// TIA Portal project "CajaDeLeche" (V14)

(* hardware
DEVICE "S71500/ET200MP-Station_1"  S7-1500 station
   slot 0: "Profilschiene_0"  6ES7 590-1***0-0AA0
   slot 1: "PLC_1"  CPU 1511-1 PN  6ES7 511-1AK00-0AB0  V1.8
   slot 2: "AI 8xU/I/RTD/TC ST_1"  AI 8xU/I/RTD/TC ST  6ES7 531-7KF00-0AB0  V2.0
   slot 3: "AI 8xU/I/RTD/TC ST_2"  AI 8xU/I/RTD/TC ST  6ES7 531-7KF00-0AB0  V2.0
   slot 4: "AI 8xU/I/RTD/TC ST_3"  AI 8xU/I/RTD/TC ST  6ES7 531-7KF00-0AB0  V2.0
   slot 5: "AI 4xU/I/RTD/TC ST_1"  AI 4xU/I/RTD/TC ST  6ES7 531-7QD00-0AB0  V1.0
   slot 6: "DI 32x24VDC BA_1"  DI 32x24VDC BA  6ES7 521-1BL10-0AA0  V1.0
   slot 7: "DI 32x24VDC BA_2"  DI 32x24VDC BA  6ES7 521-1BL10-0AA0  V1.0
   slot 8: "AQ 4xU/I ST_1"  AQ 4xU/I ST  6ES7 532-5HD00-0AB0  V2.1
   slot 9: "DI 16x24VDC BA_1"  DI 16x24VDC BA  6ES7 521-1BH10-0AA0  V1.0
   slot 10: "DQ 32x24VDC/0.5A ST_1"  DQ 32x24VDC/0.5A ST  6ES7 522-1BL00-0AB0  V2.0
   slot 11: "AQ 4xU/I ST_2"  AQ 4xU/I ST  6ES7 532-5HD00-0AB0  V2.1
   slot 12: "AQ 4xU/I ST_3"  AQ 4xU/I ST  6ES7 532-5HD00-0AB0  V2.1
DEVICE "PC-System_2"  SIMATIC PC station
   slot 0: "Estación PC SIMATIC"  Rail  SIMATIC PC-Station  V1.0
      slot 125: "Stationmanager"  Station_Manager  V6.0.4
   slot 1: "HMI_RT_1"  WinCC RT Professional  6AV2 105-0xxxx-xxxx  14.0.1.0
   slot 2: "IE general_1"  IE General  IE_CP  V8.2.0
*)

// ===== PLC "PLC_1"  CPU 1511-1 PN =====

VAR_GLOBAL   // PLC tag table "Standard-Variablentabelle"
   "Tag_1" AT %E0.0 : Bool;
   "Tag_2" AT %A0.0 : Bool;
   "Tag_3" AT %E0.1 : Bool;
   "LCV001" AT %QW0 : Int;
   "FCV001" AT %QW2 : Int;
   "LT001" AT %IW0 : Int;
   "FT001" AT %IW2 : Int;
   "S_Arranque" AT %I56.0 : Bool;
   "S_Parada" AT %I56.1 : Bool;
   "B_Reset" AT %I56.2 : Bool;
   "SD010" AT %I56.3 : Bool;
   "SD020" AT %I56.4 : Bool;   // Detecta la presencia de la caja vacia
   "SD021" AT %I56.5 : Bool;   // Detecta la presencia de la caja cuando se esta llenando
   "Emisor_Cajas" AT %Q8.0 : Bool;
   "MZ020" AT %Q8.1 : Bool;   // Movimiento Eje Z
   "SZ020" AT %Q8.2 : Bool;   // Succion
   "MZ030" AT %Q8.3 : Bool;   // Movimiento Eje Z
   "SZ030" AT %Q8.4 : Bool;   // Succion
   "CINTA1" AT %Q8.5 : Bool;
   "CINTA2" AT %Q8.6 : Bool;
   "CINTA3" AT %Q8.7 : Bool;
   "CINTA4" AT %Q9.0 : Bool;
   "BSTOP1" AT %Q9.1 : Bool;
   "SD030" AT %I56.7 : Bool;   // Detecta la presencia de la caja llena
   "SD031" AT %I57.0 : Bool;   // Detecta la presencia de la caja cuando se esta colocando la tapa
   "SD022" AT %I56.6 : Bool;
   "SD032" AT %I57.1 : Bool;
   "SD040" AT %I57.2 : Bool;
   "BARRERA_IR" AT %IW4 : Int;
   "Tag_4" AT %QB0 : Byte;
   "Tag_5" AT %QB8 : Byte;
   "Tag_6" AT %QB9 : Byte;
   "Tag_7" AT %QB10 : Byte;
   "Display" AT %QW6 : Int;
   "V001" AT %Q11.2 : Bool;
   "WL04" AT %Q11.3 : Bool;
   "BSTOP2" AT %Q9.2 : Bool;
   "LedBajoNivel" AT %Q9.3 : Bool;
   "LedNivelOk" AT %Q9.4 : Bool;
   "LedContador" AT %Q9.5 : Bool;
   "LedFin" AT %Q9.6 : Bool;
   "LedLLenado" AT %Q9.7 : Bool;
   "VPISTON" AT %QW12 : Int;
   "DISPLAY_NIVEL_TANQUE" AT %QW14 : Int;
   "DISPLAY_SET_NIVEL" AT %QW16 : Int;
   "DISPLAY_NUMERO_BOTELLAS" AT %QW18 : Int;
   "DISPLAY_CONTADOR" AT %QW20 : Int;
   "DISPLAY_PID" AT %QW22 : Int;
   "DISPLAY_SETPINT_LITROS" AT %QW24 : Int;
   "P_PISTON" AT %IW8 : Int;
   "POTE_NIVEL" AT %IW10 : Int;
   "POTE_CANTIDAD_BOTELLA" AT %IW12 : Int;
   "POTE_ESTABLECER_LITROS" AT %IW14 : Int;
   "B_Remoto" AT %I57.3 : Bool;
   "B_Local" AT %I57.4 : Bool;
   "B_Formula1" AT %I57.5 : Bool;
   "B_Formula 2" AT %I57.6 : Bool;
END_VAR

VAR_GLOBAL   // PLC tag table "Paletizado"
   "CINTA_SUPERIOR" AT %Q10.0 : Bool;
   "LIMITE_EMPUJADOR" AT %I57.7 : Bool;
   "PALETA" AT %Q10.1 : Bool;
   "EMPUJADOR" AT %Q10.2 : Bool;
   "LIMITE_PLACA" AT %I58.0 : Bool;
   "PLACA" AT %Q10.3 : Bool;
   "EMISOR_PALLET" AT %Q10.4 : Bool;
   "SENSOR_REFLECTIVO_TRASERO" AT %I58.1 : Bool;
   "SENSOR_REFLECTIVO_DELANTERO" AT %I58.2 : Bool;
   "TRANSPORTADOR_DE_RODILLOS_1" AT %Q10.5 : Bool;
   "SENSOR_LIMITE_FRONTAL" AT %I58.3 : Bool;
   "SENSOR_LIMITE_TRASERO" AT %I58.4 : Bool;
   "CADENA_PALETIZADORA" AT %Q10.6 : Bool;
   "ELEVADOR_SUBIR" AT %Q10.7 : Bool;
   "ELEVADOR_BAJAR" AT %Q11.0 : Bool;
   "ELEVADOR_MOVER_AL_LIMITE" AT %Q11.1 : Bool;
   "SENSOR_CONTADOR" AT %I58.5 : Bool;
   "JUNTAR" AT %Q11.4 : Bool;
   "SENSOR_LIMITE_ELEVADOR" AT %I58.6 : Bool;
END_VAR

DATA_BLOCK "Datos"   // DB1
{ S7_Optimized_Access := 'TRUE' }
VERSION : 0.1
   VAR
      Lecturas : Struct
         "LT001 (mm)" : Real;
         "VT001(L)" : Int;
         "LT001F (mm)" : Real;
         NCAJAS : Int;
         "FT001 (m3/s)" : Real;
         "Posicion (cm)" : Real;
         "Velocidad (cm/s)" : Int;
      END_STRUCT;
      "Set Point" : Struct
         SetPoint_Litros : Int := 1000;
         SetPoint_Cantidad : Int := 20;
         SetPoint_LCV001 : Int := 2000;
      END_STRUCT;
      Dispositivos : Struct
         Tanque : Struct
            L_Maximo : Real := 3000.0;
            L_Minimo : Real;
         END_STRUCT;
      END_STRUCT;
      Constantes : Struct
         A_Lectura_Max_10V : Int := 27648;
         A_Lectura_Min_0V : Int;
      END_STRUCT;
      Etiquetas : Struct
         Emisor : Struct
            Marca : Array[0..10] of Bool;
         END_STRUCT;
         LlenarBotella : Bool;
         Reset : Bool;
         Proceso : Struct
            On : Bool;
            Off : Bool;
         END_STRUCT;
      END_STRUCT;
   END_VAR
BEGIN
END_DATA_BLOCK

DATA_BLOCK "Tableros_DB"   // DB4
{ S7_Optimized_Access := 'TRUE' }
VERSION : 0.1
// stored: InstanceOfName Tableros
"Tableros"
BEGIN
END_DATA_BLOCK

DATA_BLOCK "Paletizado_DB"   // DB5
{ S7_Optimized_Access := 'TRUE' }
VERSION : 0.1
// stored: InstanceOfName Paletizado
"Paletizado"
BEGIN
END_DATA_BLOCK

DATA_BLOCK "Integrador_DB"   // DB14
{ S7_Optimized_Access := 'TRUE' }
VERSION : 0.1
// stored: InstanceOfName Integrador
"Integrador"
BEGIN
END_DATA_BLOCK

DATA_BLOCK "Proceso_Linea_DB"   // DB22
{ S7_Optimized_Access := 'TRUE' }
VERSION : 0.1
// stored: InstanceOfName Proceso_Linea
"Proceso_Linea"
BEGIN
END_DATA_BLOCK

// folder: System blocks/Program resources

DATA_BLOCK "Empujador_retardo"   // DB6
{ S7_Optimized_Access := 'TRUE' }
AUTHOR : Simatic
FAMILY : IEC
NAME : IEC_TMR
VERSION : 1.0
// stored: InstanceOfName IEC_TIMER
"IEC_TIMER"
BEGIN
END_DATA_BLOCK

DATA_BLOCK "Tiempo_Emisor_Pallet"   // DB7
{ S7_Optimized_Access := 'TRUE' }
AUTHOR : Simatic
FAMILY : IEC
NAME : IEC_TMR
VERSION : 1.0
// stored: InstanceOfName IEC_TIMER
"IEC_TIMER"
BEGIN
END_DATA_BLOCK

DATA_BLOCK "RETARDO"   // DB8
{ S7_Optimized_Access := 'TRUE' }
AUTHOR : Simatic
FAMILY : IEC
NAME : IEC_TMR
VERSION : 1.0
// stored: InstanceOfName IEC_TIMER
"IEC_TIMER"
BEGIN
END_DATA_BLOCK

DATA_BLOCK "BAJAR"   // DB9
{ S7_Optimized_Access := 'TRUE' }
AUTHOR : Simatic
FAMILY : IEC
NAME : IEC_TMR
VERSION : 1.0
// stored: InstanceOfName IEC_TIMER
"IEC_TIMER"
BEGIN
END_DATA_BLOCK

DATA_BLOCK "Contador_Cajas_Paletizadora_A"   // DB10
{ S7_Optimized_Access := 'TRUE' }
AUTHOR : Simatic
FAMILY : IEC
NAME : CNTR
VERSION : 1.0
// stored: InstanceOfName IEC_COUNTER
"IEC_COUNTER"
BEGIN
END_DATA_BLOCK

DATA_BLOCK "Contar_3_Filas"   // DB11
{ S7_Optimized_Access := 'TRUE' }
AUTHOR : Simatic
FAMILY : IEC
NAME : CNTR
VERSION : 1.0
// stored: InstanceOfName IEC_COUNTER
"IEC_COUNTER"
BEGIN
END_DATA_BLOCK

DATA_BLOCK "iee"   // DB12
{ S7_Optimized_Access := 'TRUE' }
AUTHOR : Simatic
FAMILY : IEC
NAME : CNTR
VERSION : 1.0
// stored: InstanceOfName IEC_COUNTER
"IEC_COUNTER"
BEGIN
END_DATA_BLOCK

DATA_BLOCK "RETARDO_BAJAR_PALLET"   // DB13
{ S7_Optimized_Access := 'TRUE' }
AUTHOR : Simatic
FAMILY : IEC
NAME : IEC_TMR
VERSION : 1.0
// stored: InstanceOfName IEC_TIMER
"IEC_TIMER"
BEGIN
END_DATA_BLOCK

DATA_BLOCK "Emisor"   // DB18
{ S7_Optimized_Access := 'TRUE' }
AUTHOR : Simatic
FAMILY : IEC
NAME : IEC_TMR
VERSION : 1.0
// stored: InstanceOfName IEC_TIMER
"IEC_TIMER"
BEGIN
END_DATA_BLOCK

DATA_BLOCK "Ton_ColocacionDeTapa"   // DB19
{ S7_Optimized_Access := 'TRUE' }
AUTHOR : Simatic
FAMILY : IEC
NAME : IEC_TMR
VERSION : 1.0
// stored: InstanceOfName IEC_TIMER
"IEC_TIMER"
BEGIN
END_DATA_BLOCK

DATA_BLOCK "Contador_BotellasEmitidas"   // DB21
{ S7_Optimized_Access := 'TRUE' }
AUTHOR : Simatic
FAMILY : IEC
NAME : CNTR
VERSION : 1.0
// stored: InstanceOfName IEC_COUNTER
"IEC_COUNTER"
BEGIN
END_DATA_BLOCK

DATA_BLOCK "IEC_Timer_0_DB_1"   // DB26
{ S7_Optimized_Access := 'TRUE' }
AUTHOR : Simatic
FAMILY : IEC
NAME : IEC_TMR
VERSION : 1.0
// stored: InstanceOfName IEC_TIMER
"IEC_TIMER"
BEGIN
END_DATA_BLOCK

// folder: (top level)

FUNCTION_BLOCK "Tableros"   // FB1, LAD
{ S7_Optimized_Access := 'TRUE' }
VERSION : 0.1
   VAR_INPUT
      Local : Bool;
      Remoto : Bool;
      "Formula 1" : Bool;
      "Formula 2" : Bool;
      Nivel : Real;
      "Nro Botellas" : Real;
      "mL por Botella" : Real;
   END_VAR
   VAR_OUTPUT
      Display_Nivel_Actual : Int;
      Display_Nivel_Seteado : Int;
      Display_Nro_Botellas : Int;
      Display_Contador : Int;
      Display_ml : Int;
      Display_PID : Int;
   END_VAR
   VAR
      "Nivel Temp" : Int;
      "Numero Temp" : Int;
      "mL Temp" : Int;
   END_VAR
BEGIN

REGION Network 1
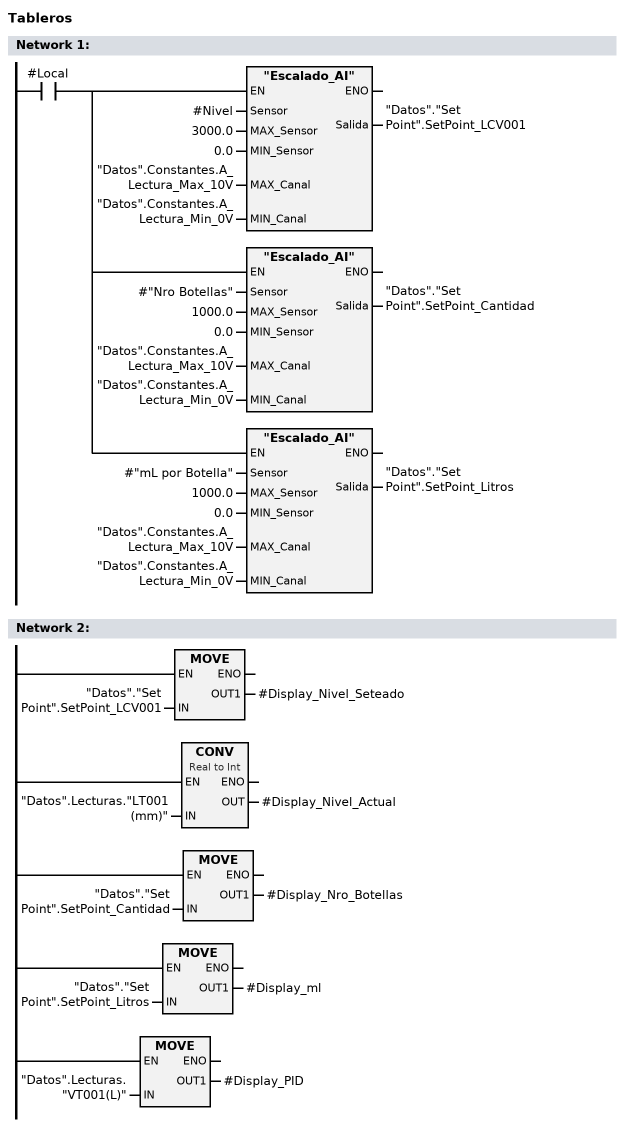
   RUNG wire#powerrail
      Contact( #Local )
      wire#w1
      "Escalado_AI"(Sensor := #Nivel, MAX_Sensor := 3000.0, MIN_Sensor := 0.0, MAX_Canal := "Datos".Constantes.A_Lectura_Max_10V, MIN_Canal := "Datos".Constantes.A_Lectura_Min_0V, Salida => "Datos"."Set Point".SetPoint_LCV001)
   END_RUNG
   RUNG wire#w1
      "Escalado_AI"(Sensor := #"Nro Botellas", MAX_Sensor := 1000.0, MIN_Sensor := 0.0, MAX_Canal := "Datos".Constantes.A_Lectura_Max_10V, MIN_Canal := "Datos".Constantes.A_Lectura_Min_0V, Salida => "Datos"."Set Point".SetPoint_Cantidad)
   END_RUNG
   RUNG wire#w1
      "Escalado_AI"(Sensor := #"mL por Botella", MAX_Sensor := 1000.0, MIN_Sensor := 0.0, MAX_Canal := "Datos".Constantes.A_Lectura_Max_10V, MIN_Canal := "Datos".Constantes.A_Lectura_Min_0V, Salida => "Datos"."Set Point".SetPoint_Litros)
   END_RUNG
   // the same network as SCL:
   IF #Local THEN
       "Escalado_AI"(Sensor := #Nivel,
                     MAX_Sensor := 3000.0,
                     MIN_Sensor := 0.0,
                     MAX_Canal := "Datos".Constantes.A_Lectura_Max_10V,
                     MIN_Canal := "Datos".Constantes.A_Lectura_Min_0V,
                     Salida => "Datos"."Set Point".SetPoint_LCV001);
       "Escalado_AI"(Sensor := #"Nro Botellas",
                     MAX_Sensor := 1000.0,
                     MIN_Sensor := 0.0,
                     MAX_Canal := "Datos".Constantes.A_Lectura_Max_10V,
                     MIN_Canal := "Datos".Constantes.A_Lectura_Min_0V,
                     Salida => "Datos"."Set Point".SetPoint_Cantidad);
       "Escalado_AI"(Sensor := #"mL por Botella",
                     MAX_Sensor := 1000.0,
                     MIN_Sensor := 0.0,
                     MAX_Canal := "Datos".Constantes.A_Lectura_Max_10V,
                     MIN_Canal := "Datos".Constantes.A_Lectura_Min_0V,
                     Salida => "Datos"."Set Point".SetPoint_Litros);
   END_IF;
END_REGION

REGION Network 2
   RUNG wire#powerrail
      Move(in := "Datos"."Set Point".SetPoint_LCV001, out1 => #Display_Nivel_Seteado)
   END_RUNG
   RUNG wire#powerrail
      { S7_Templates := "[SrcType := Real, DestType := Int]" } Convert(in := "Datos".Lecturas."LT001 (mm)", out => #Display_Nivel_Actual)
   END_RUNG
   RUNG wire#powerrail
      Move(in := "Datos"."Set Point".SetPoint_Cantidad, out1 => #Display_Nro_Botellas)
   END_RUNG
   RUNG wire#powerrail
      Move(in := "Datos"."Set Point".SetPoint_Litros, out1 => #Display_ml)
   END_RUNG
   RUNG wire#powerrail
      Move(in := "Datos".Lecturas."VT001(L)", out1 => #Display_PID)
   END_RUNG
   // the same network as SCL:
   #Display_Nivel_Seteado := "Datos"."Set Point".SetPoint_LCV001;
   #Display_Nivel_Actual := REAL_TO_INT("Datos".Lecturas."LT001 (mm)");
   #Display_Nro_Botellas := "Datos"."Set Point".SetPoint_Cantidad;
   #Display_ml := "Datos"."Set Point".SetPoint_Litros;
   #Display_PID := "Datos".Lecturas."VT001(L)";
END_REGION
END_FUNCTION_BLOCK

FUNCTION_BLOCK "Paletizado"   // FB2, LAD
{ S7_Optimized_Access := 'TRUE' }
VERSION : 0.1
   VAR_INPUT
      ARRANQUE : Bool;
      LIMITE_EMPUJADOR : Bool;
      LIMITE_PLACA : Bool;
      SENSOR_REFLECTIVO_TRASERO : Bool;
      SENSOR_REFLECTIVO_DELANTERO : Bool;
      SENSOR_LIMITE_FRONTAL : Bool;
      SENSOR_LIMITE_TRESERO : Bool;
      SENSOR_CONTADOR : Bool;
      SENSOR_LIMITE_ELEVADOR : Bool;
   END_VAR
   VAR_OUTPUT
      CINTA_SUPERIOR : Bool;
      PALETA : Bool;
      EMPUJADOR : Bool;
      PLACA : Bool;
      EMISOR_PALLET : Bool;
      TRANSPORTADOR_DE_RODILLO : Bool;
      CADENA_PALETIZADORA : Bool;
      ELEVADOR_SUBIR : Bool;
      ELEVADOR_BAJAR : Bool;
      ELEVADOR_MOVER_AL_LIMITE : Bool;
      JUNTAR : Bool;
   END_VAR
   VAR
      Flanco : Array[0..40] of Bool;
      Marcas : Array[0..10] of Bool;
      Marca_Emisor : Array[0..10] of Bool;
      REINICIAR_CONT_A : Bool;
      "Contar 2 CAJAS" : Int;
      FILAS : Bool := true;
      CONTEO_B : Int := 2;
      REINICIAR_CONTEO_B : Bool;
      CONTEO_A : Int := 3;
      REINICIAR_CONTEO_C : Bool;
      BYTES : Byte := 16#0;
      CONTAR_ALTURA_FILAS : Bool;
   END_VAR
   VAR_TEMP   // added for the SCL form of the ladder/FBD networks
      _w1 : Bool;
      _w2 : Bool;
      _w3 : Bool;
      _w4 : Bool;
      _w5 : Bool;
   END_VAR
BEGIN

REGION Network 1: Movimiento del Pallet
   // Movimiento del ascensor del Palletizador.
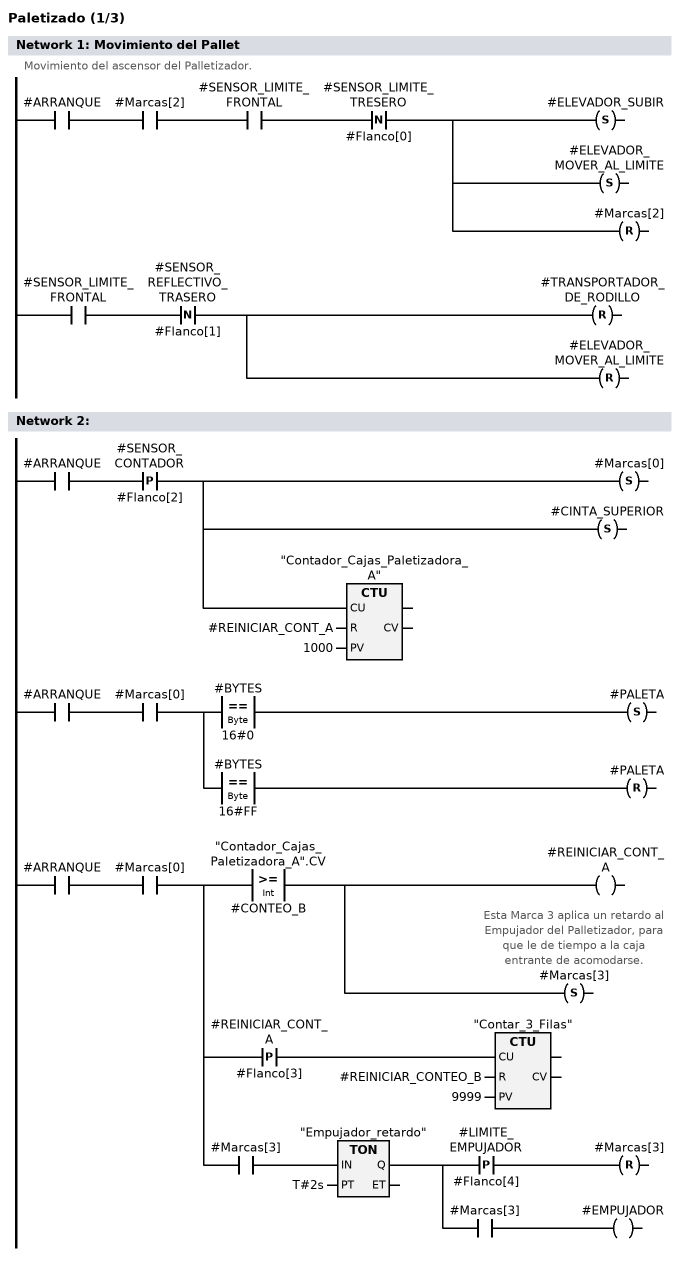
   RUNG wire#powerrail
      Contact( #ARRANQUE )
      Contact( #Marcas[2] )
      Contact( #SENSOR_LIMITE_FRONTAL )
      N_Contact(operand := #SENSOR_LIMITE_TRESERO, bit := #Flanco[0])
      wire#w1
      S_Coil( #ELEVADOR_SUBIR )
   END_RUNG
   RUNG wire#w1
      S_Coil( #ELEVADOR_MOVER_AL_LIMITE )
   END_RUNG
   RUNG wire#w1
      R_Coil( #Marcas[2] )
   END_RUNG
   RUNG wire#powerrail
      Contact( #SENSOR_LIMITE_FRONTAL )
      N_Contact(operand := #SENSOR_REFLECTIVO_TRASERO, bit := #Flanco[1])
      wire#w2
      R_Coil( #TRANSPORTADOR_DE_RODILLO )
   END_RUNG
   RUNG wire#w2
      R_Coil( #ELEVADOR_MOVER_AL_LIMITE )
   END_RUNG
   // the same network as SCL:
   #_w1 := #ARRANQUE AND #Marcas[2] AND #SENSOR_LIMITE_FRONTAL AND NOT #SENSOR_LIMITE_TRESERO AND #Flanco[0];   // falling edge of #SENSOR_LIMITE_TRESERO
   #Flanco[0] := #SENSOR_LIMITE_TRESERO;
   IF #_w1 THEN
       #ELEVADOR_SUBIR := TRUE;
       #ELEVADOR_MOVER_AL_LIMITE := TRUE;
       #Marcas[2] := FALSE;
   END_IF;
   #_w2 := #SENSOR_LIMITE_FRONTAL AND NOT #SENSOR_REFLECTIVO_TRASERO AND #Flanco[1];   // falling edge of #SENSOR_REFLECTIVO_TRASERO
   #Flanco[1] := #SENSOR_REFLECTIVO_TRASERO;
   IF #_w2 THEN
       #TRANSPORTADOR_DE_RODILLO := FALSE;
       #ELEVADOR_MOVER_AL_LIMITE := FALSE;
   END_IF;
END_REGION

REGION Network 2
   #_w1 := #ARRANQUE AND #SENSOR_CONTADOR AND NOT #Flanco[2];   // rising edge of #SENSOR_CONTADOR
   #Flanco[2] := #SENSOR_CONTADOR;
   IF #_w1 THEN
       #Marcas[0] := TRUE;
       #CINTA_SUPERIOR := TRUE;
   END_IF;
   "Contador_Cajas_Paletizadora_A".CTU(CU := #_w1, R := #REINICIAR_CONT_A, PV := 1000);
   #_w2 := #ARRANQUE AND #Marcas[0];
   IF #_w2 AND (#BYTES = 16#0) THEN #PALETA := TRUE; END_IF;
   IF #_w2 AND (#BYTES = 16#FF) THEN #PALETA := FALSE; END_IF;
   #_w3 := #ARRANQUE AND #Marcas[0];
   #REINICIAR_CONT_A := #_w3 AND ("Contador_Cajas_Paletizadora_A".CV >= #CONTEO_B);
   IF #REINICIAR_CONT_A THEN
       #Marcas[3] := TRUE;   // Esta Marca 3 aplica un retardo al Empujador del Palletizador, para que le de tiempo a la caja entrante de acomodarse.
   END_IF;
   #_w4 := #_w3 AND #REINICIAR_CONT_A AND NOT #Flanco[3];   // rising edge of #REINICIAR_CONT_A
   #Flanco[3] := #REINICIAR_CONT_A;
   "Contar_3_Filas".CTU(CU := #_w4, R := #REINICIAR_CONTEO_B, PV := 9999);
   "Empujador_retardo".TON(IN := #_w3 AND #Marcas[3], PT := T#2s);
   #_w5 := "Empujador_retardo".Q AND #LIMITE_EMPUJADOR AND NOT #Flanco[4];   // rising edge of #LIMITE_EMPUJADOR
   #Flanco[4] := #LIMITE_EMPUJADOR;
   IF #_w5 THEN #Marcas[3] := FALSE; END_IF;
   #EMPUJADOR := "Empujador_retardo".Q AND #Marcas[3];
END_REGION

REGION Network 3
   // Colocacion de las Cajas en el Pallet
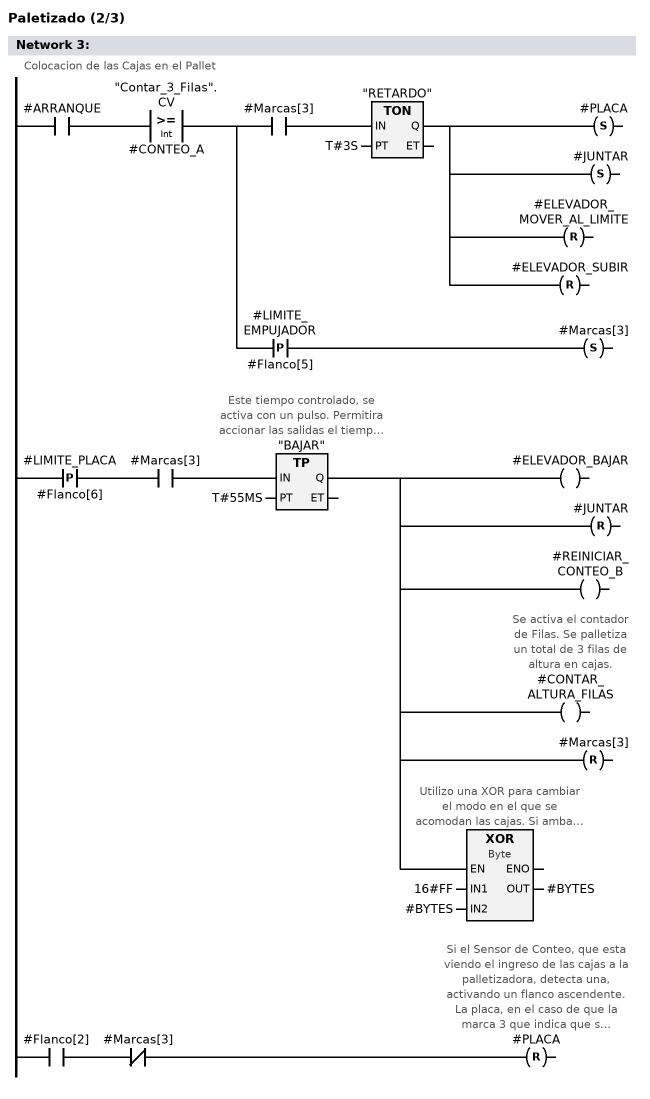
   // no checked SCL form for this network; see the picture
END_REGION

REGION Network 4
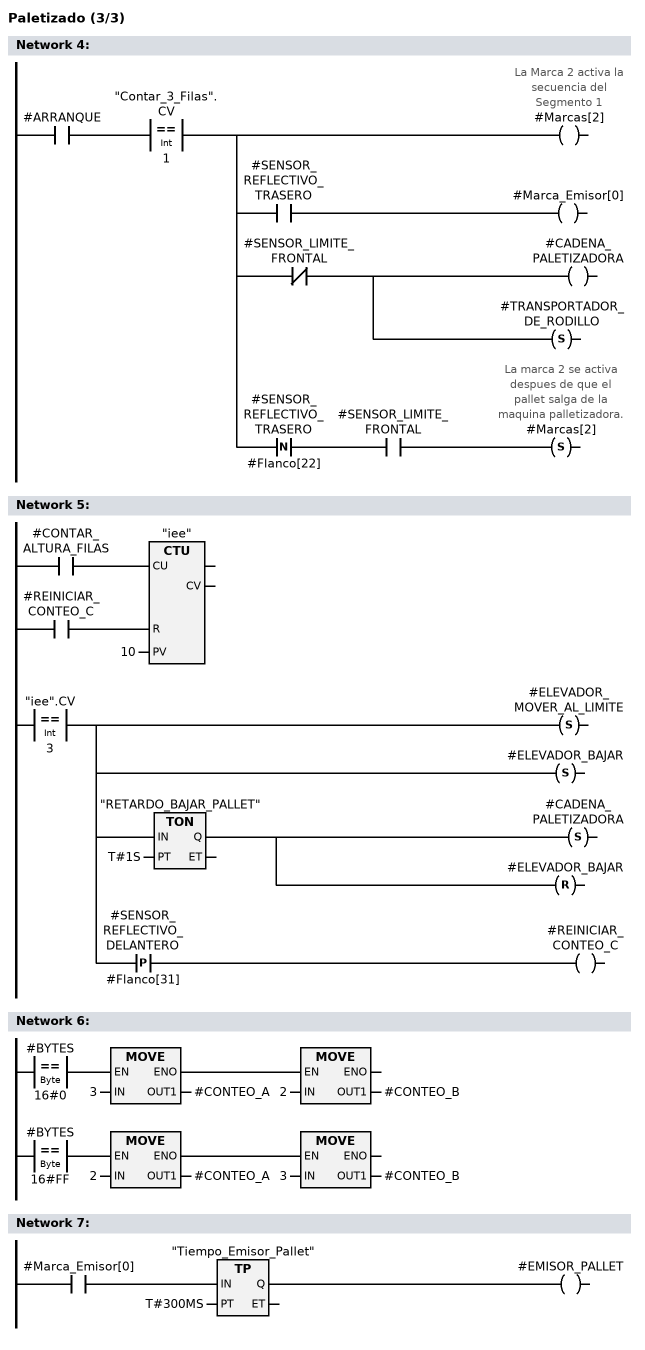
   RUNG wire#powerrail
      Contact( #ARRANQUE )
      { S7_Templates := "SrcType := Int" } EQ_Contact(in1 := "Contar_3_Filas".CV, in2 := 1)
      wire#w1
      Coil( #Marcas[2] )   // La Marca 2 activa la secuencia del Segmento 1
   END_RUNG
   RUNG wire#w1
      Contact( #SENSOR_REFLECTIVO_TRASERO )
      Coil( #Marca_Emisor[0] )
   END_RUNG
   RUNG wire#w1
      I_Contact( #SENSOR_LIMITE_FRONTAL )
      wire#w2
      Coil( #CADENA_PALETIZADORA )
   END_RUNG
   RUNG wire#w2
      S_Coil( #TRANSPORTADOR_DE_RODILLO )
   END_RUNG
   RUNG wire#w1
      N_Contact(operand := #SENSOR_REFLECTIVO_TRASERO, bit := #Flanco[22])
      Contact( #SENSOR_LIMITE_FRONTAL )
      S_Coil( #Marcas[2] )   // La marca 2 se activa despues de que el pallet salga de la maquina palletizadora.
   END_RUNG
   // the same network as SCL:
   #Marcas[2] := #ARRANQUE AND ("Contar_3_Filas".CV = 1);   // La Marca 2 activa la secuencia del Segmento 1
   #Marca_Emisor[0] := #ARRANQUE AND ("Contar_3_Filas".CV = 1) AND #SENSOR_REFLECTIVO_TRASERO;
   #CADENA_PALETIZADORA := #ARRANQUE AND ("Contar_3_Filas".CV = 1) AND NOT #SENSOR_LIMITE_FRONTAL;
   IF #CADENA_PALETIZADORA THEN #TRANSPORTADOR_DE_RODILLO := TRUE; END_IF;
   #_w1 := #ARRANQUE AND ("Contar_3_Filas".CV = 1) AND NOT #SENSOR_REFLECTIVO_TRASERO AND #Flanco[22];   // falling edge of #SENSOR_REFLECTIVO_TRASERO
   #Flanco[22] := #SENSOR_REFLECTIVO_TRASERO;
   IF #_w1 AND #SENSOR_LIMITE_FRONTAL THEN
       #Marcas[2] := TRUE;   // La marca 2 se activa despues de que el pallet salga de la maquina palletizadora.
   END_IF;
END_REGION

REGION Network 5
   "iee".CTU(CU := #CONTAR_ALTURA_FILAS, R := #REINICIAR_CONTEO_C, PV := 10);
   #_w1 := "iee".CV = 3;
   IF #_w1 THEN
       #ELEVADOR_MOVER_AL_LIMITE := TRUE;
       #ELEVADOR_BAJAR := TRUE;
   END_IF;
   "RETARDO_BAJAR_PALLET".TON(IN := #_w1, PT := T#1S);
   IF "RETARDO_BAJAR_PALLET".Q THEN
       #CADENA_PALETIZADORA := TRUE;
       #ELEVADOR_BAJAR := FALSE;
   END_IF;
   #_w2 := #_w1 AND #SENSOR_REFLECTIVO_DELANTERO AND NOT #Flanco[31];   // rising edge of #SENSOR_REFLECTIVO_DELANTERO
   #Flanco[31] := #SENSOR_REFLECTIVO_DELANTERO;
   #REINICIAR_CONTEO_C := #_w2;
END_REGION

REGION Network 6
   RUNG wire#powerrail
      { S7_Templates := "SrcType := Byte" } EQ_Contact(in1 := #BYTES, in2 := 16#0)
      Move(in := 3, out1 => #CONTEO_A)
      Move(in := 2, out1 => #CONTEO_B)
   END_RUNG
   RUNG wire#powerrail
      { S7_Templates := "SrcType := Byte" } EQ_Contact(in1 := #BYTES, in2 := 16#FF)
      Move(in := 2, out1 => #CONTEO_A)
      Move(in := 3, out1 => #CONTEO_B)
   END_RUNG
   // the same network as SCL:
   IF #BYTES = 16#0 THEN
       #CONTEO_A := 3;
       #CONTEO_B := 2;
   END_IF;
   IF #BYTES = 16#FF THEN
       #CONTEO_A := 2;
       #CONTEO_B := 3;
   END_IF;
END_REGION

REGION Network 7
   "Tiempo_Emisor_Pallet".TP(IN := #Marca_Emisor[0], PT := T#300MS);
   #EMISOR_PALLET := "Tiempo_Emisor_Pallet".Q;
END_REGION
END_FUNCTION_BLOCK

FUNCTION_BLOCK "Integrador"   // FB5, LAD
{ S7_Optimized_Access := 'TRUE' }
VERSION : 0.1
   VAR_INPUT
      Señal : Real;
      Tm : Real;
      Reset : Bool;
   END_VAR
   VAR_OUTPUT
      Integracion : Int;
   END_VAR
   VAR
      Almacenamiento : Real;
      Multiplicacion : Real;
      Cero : Real := 0.0;
      Temporal : Real;
   END_VAR
BEGIN

REGION Network 1
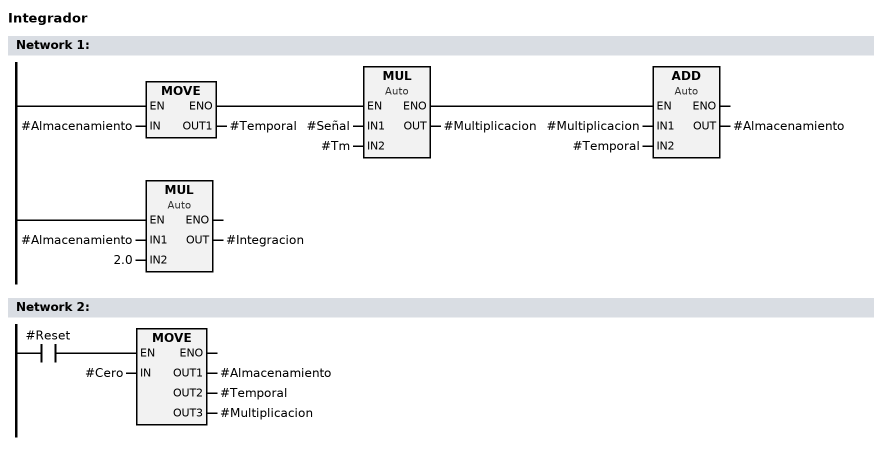
   RUNG wire#powerrail
      Move(in := #Almacenamiento, out1 => #Temporal)
      Mul(in1 := #Señal, in2 := #Tm, out => #Multiplicacion)
      Add(in1 := #Multiplicacion, in2 := #Temporal, out => #Almacenamiento)
   END_RUNG
   RUNG wire#powerrail
      Mul(in1 := #Almacenamiento, in2 := 2.0, out => #Integracion)
   END_RUNG
   // the same network as SCL:
   #Temporal := #Almacenamiento;
   #Multiplicacion := #Señal * #Tm;
   #Almacenamiento := #Multiplicacion + #Temporal;
   #Integracion := #Almacenamiento * 2.0;
END_REGION

REGION Network 2
   RUNG wire#powerrail
      Contact( #Reset )
      Move(in := #Cero, out1 => #Almacenamiento, out2 => #Temporal, out3 => #Multiplicacion)
   END_RUNG
   // the same network as SCL:
   IF #Reset THEN
       #Almacenamiento := #Cero;
       #Temporal := #Cero;
       #Multiplicacion := #Cero;
   END_IF;
END_REGION
END_FUNCTION_BLOCK

FUNCTION_BLOCK "Proceso_Linea"   // FB6, LAD
{ S7_Optimized_Access := 'TRUE' }
VERSION : 0.1
   VAR_INPUT
      Arranque : Bool;
      Parada : Bool;
      "Parada de Emergencia" : Bool;
      "Nivel Tanque (mm)" : Real;
      "Caudal (m3/s)" : Real;
      "Volumen (l)" : Real;
      "Receta 1" : Bool;
      "Receta 2" : Bool;
      SD010 : Bool;
      SD020 : Bool;
      SD021 : Bool;
      SD022 : Bool;
      SD030 : Bool;
      SD031 : Bool;
      SD032 : Bool;
      SD040 : Bool;
      "Posicion Piston" : Real;
   END_VAR
   VAR_OUTPUT
      LED_NIVEL_BAJO : Bool;
      LED_NIVEL_OK : Bool;
      LED_CONTEO_ON : Bool;
      LED_PROCESO_FINALIZADO : Bool;
      LED_LLENADO : Bool;
      Alarma : Bool;
      "Barrera 1" : Bool;
      "Barrera 2" : Bool;
      "Velocidad Piston" : Int;
      "Movimento Eje Z 020" : Bool;
      "Succion 020" : Bool;
      "Movimiento Eje Z 030" : Bool;
      "Succion 030" : Bool;
      Emisor : Bool;
      "Cinta 1" : Bool;
      "Cinta 2" : Bool;
      "Cinta 3" : Bool;
      "Cinta 4" : Bool;
      Display : Int;
      "Resetear Volumen" : Bool;
   END_VAR
   VAR
      Paso : Array[0..10] of Bool;
      Marca : Array[0..10] of Bool;
      Min_Litros : Real;
      Max_Litros : Real;
      Emitir : Array[0..2] of Bool;
      Flanco : Array[0..20] of Bool;
   END_VAR
   VAR RETAIN
      Estados : Array[0..20] of Bool;
   END_VAR
   VAR
      "Byte" : Array[0..20] of Byte;
      Contador_Emisor : Int;
   END_VAR
   VAR_TEMP   // added for the SCL form of the ladder/FBD networks
      _w1 : Bool;
      _w2 : Bool;
      _w3 : Bool;
      _w4 : Bool;
   END_VAR
BEGIN

REGION Network 1: Arranque
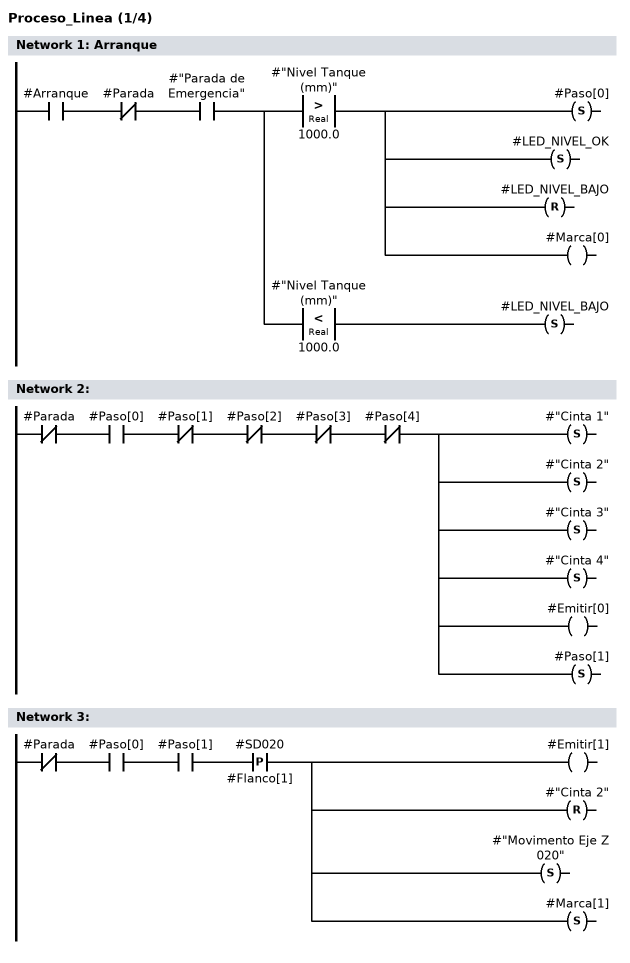
   RUNG wire#powerrail
      Contact( #Arranque )
      I_Contact( #Parada )
      Contact( #"Parada de Emergencia" )
      wire#w1
      { S7_Templates := "SrcType := Real" } GT_Contact(in1 := #"Nivel Tanque (mm)", in2 := 1000.0)
      wire#w2
      S_Coil( #Paso[0] )
   END_RUNG
   RUNG wire#w2
      S_Coil( #LED_NIVEL_OK )
   END_RUNG
   RUNG wire#w2
      R_Coil( #LED_NIVEL_BAJO )
   END_RUNG
   RUNG wire#w2
      Coil( #Marca[0] )
   END_RUNG
   RUNG wire#w1
      { S7_Templates := "SrcType := Real" } LT_Contact(in1 := #"Nivel Tanque (mm)", in2 := 1000.0)
      S_Coil( #LED_NIVEL_BAJO )
   END_RUNG
   // the same network as SCL:
   #_w1 := #Arranque AND NOT #Parada AND #"Parada de Emergencia";
   #_w2 := #_w1 AND (#"Nivel Tanque (mm)" > 1000.0);
   IF #_w2 THEN
       #Paso[0] := TRUE;
       #LED_NIVEL_OK := TRUE;
       #LED_NIVEL_BAJO := FALSE;
   END_IF;
   #Marca[0] := #_w2;
   IF #_w1 AND (#"Nivel Tanque (mm)" < 1000.0) THEN #LED_NIVEL_BAJO := TRUE; END_IF;
END_REGION

REGION Network 2
   RUNG wire#powerrail
      I_Contact( #Parada )
      Contact( #Paso[0] )
      I_Contact( #Paso[1] )
      I_Contact( #Paso[2] )
      I_Contact( #Paso[3] )
      I_Contact( #Paso[4] )
      wire#w1
      S_Coil( #"Cinta 1" )
   END_RUNG
   RUNG wire#w1
      S_Coil( #"Cinta 2" )
   END_RUNG
   RUNG wire#w1
      S_Coil( #"Cinta 3" )
   END_RUNG
   RUNG wire#w1
      S_Coil( #"Cinta 4" )
   END_RUNG
   RUNG wire#w1
      Coil( #Emitir[0] )
   END_RUNG
   RUNG wire#w1
      S_Coil( #Paso[1] )
   END_RUNG
   // the same network as SCL:
   #_w1 := NOT #Parada AND #Paso[0] AND NOT #Paso[1] AND NOT #Paso[2] AND NOT #Paso[3] AND NOT #Paso[4];
   IF #_w1 THEN
       #"Cinta 1" := TRUE;
       #"Cinta 2" := TRUE;
       #"Cinta 3" := TRUE;
       #"Cinta 4" := TRUE;
   END_IF;
   #Emitir[0] := #_w1;
   IF #_w1 THEN #Paso[1] := TRUE; END_IF;
END_REGION

REGION Network 3
   RUNG wire#powerrail
      I_Contact( #Parada )
      Contact( #Paso[0] )
      Contact( #Paso[1] )
      P_Contact(operand := #SD020, bit := #Flanco[1])
      wire#w1
      Coil( #Emitir[1] )
   END_RUNG
   RUNG wire#w1
      R_Coil( #"Cinta 2" )
   END_RUNG
   RUNG wire#w1
      S_Coil( #"Movimento Eje Z 020" )
   END_RUNG
   RUNG wire#w1
      S_Coil( #Marca[1] )
   END_RUNG
   // the same network as SCL:
   #_w1 := NOT #Parada AND #Paso[0] AND #Paso[1] AND #SD020 AND NOT #Flanco[1];   // rising edge of #SD020
   #Flanco[1] := #SD020;
   #Emitir[1] := #_w1;
   IF #_w1 THEN
       #"Cinta 2" := FALSE;
       #"Movimento Eje Z 020" := TRUE;
       #Marca[1] := TRUE;
   END_IF;
END_REGION

REGION Network 4
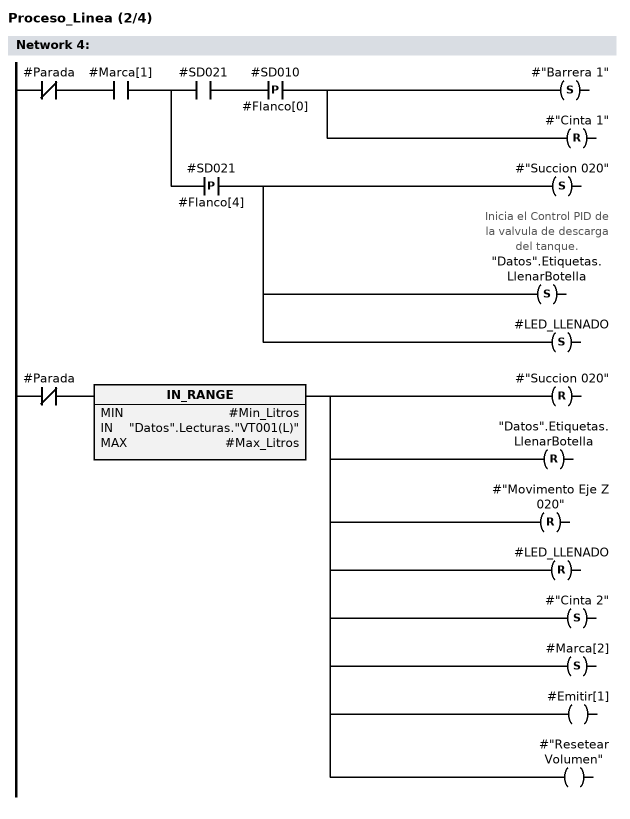
   RUNG wire#powerrail
      I_Contact( #Parada )
      Contact( #Marca[1] )
      wire#w1
      Contact( #SD021 )
      P_Contact(operand := #SD010, bit := #Flanco[0])
      wire#w2
      S_Coil( #"Barrera 1" )
   END_RUNG
   RUNG wire#w2
      R_Coil( #"Cinta 1" )
   END_RUNG
   RUNG wire#w1
      P_Contact(operand := #SD021, bit := #Flanco[4])
      wire#w3
      S_Coil( #"Succion 020" )
   END_RUNG
   RUNG wire#w3
      S_Coil( "Datos".Etiquetas.LlenarBotella )   // Inicia el Control PID de la valvula de descarga del tanque.
   END_RUNG
   RUNG wire#w3
      S_Coil( #LED_LLENADO )
   END_RUNG
   RUNG wire#powerrail
      I_Contact( #Parada )
      { S7_Templates := "SrcType := Real" } InRange(min := #Min_Litros, in := "Datos".Lecturas."VT001(L)", max := #Max_Litros)
      wire#w4
      R_Coil( #"Succion 020" )
   END_RUNG
   RUNG wire#w4
      R_Coil( "Datos".Etiquetas.LlenarBotella )
   END_RUNG
   RUNG wire#w4
      R_Coil( #"Movimento Eje Z 020" )
   END_RUNG
   RUNG wire#w4
      R_Coil( #LED_LLENADO )
   END_RUNG
   RUNG wire#w4
      S_Coil( #"Cinta 2" )
   END_RUNG
   RUNG wire#w4
      S_Coil( #Marca[2] )
   END_RUNG
   RUNG wire#w4
      Coil( #Emitir[1] )
   END_RUNG
   RUNG wire#w4
      Coil( #"Resetear Volumen" )
   END_RUNG
   // the same network as SCL:
   #_w1 := NOT #Parada AND #Marca[1];
   #_w2 := #_w1 AND #SD021 AND #SD010 AND NOT #Flanco[0];   // rising edge of #SD010
   #Flanco[0] := #SD010;
   IF #_w2 THEN
       #"Barrera 1" := TRUE;
       #"Cinta 1" := FALSE;
   END_IF;
   #_w3 := #_w1 AND #SD021 AND NOT #Flanco[4];   // rising edge of #SD021
   #Flanco[4] := #SD021;
   IF #_w3 THEN
       #"Succion 020" := TRUE;
       "Datos".Etiquetas.LlenarBotella := TRUE;   // Inicia el Control PID de la valvula de descarga del tanque.
       #LED_LLENADO := TRUE;
   END_IF;
   #_w4 := NOT #Parada AND (#Min_Litros <= "Datos".Lecturas."VT001(L)") AND ("Datos".Lecturas."VT001(L)" <= #Max_Litros);
   IF #_w4 THEN
       #"Succion 020" := FALSE;
       "Datos".Etiquetas.LlenarBotella := FALSE;
       #"Movimento Eje Z 020" := FALSE;
       #LED_LLENADO := FALSE;
       #"Cinta 2" := TRUE;
       #Marca[2] := TRUE;
   END_IF;
   #Emitir[1] := #_w4;
   #"Resetear Volumen" := #_w4;
END_REGION

REGION Network 5
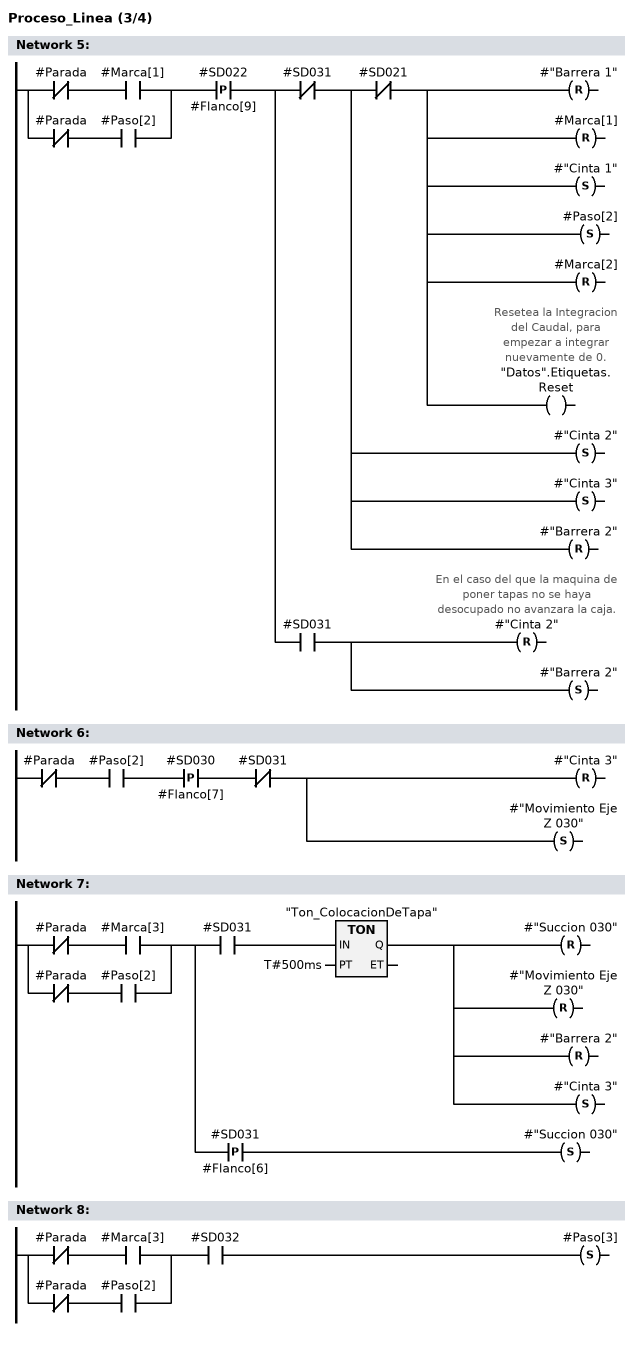
   RUNG wire#powerrail
      I_Contact( #Parada )
      Contact( #Marca[1] )
      wire#w1
      P_Contact(operand := #SD022, bit := #Flanco[9])
      wire#w2
      I_Contact( #SD031 )
      wire#w3
      I_Contact( #SD021 )
      wire#w4
      R_Coil( #"Barrera 1" )
   END_RUNG
   RUNG wire#powerrail
      I_Contact( #Parada )
      Contact( #Paso[2] )
   END_RUNG wire#w1
   RUNG wire#w4
      R_Coil( #Marca[1] )
   END_RUNG
   RUNG wire#w4
      S_Coil( #"Cinta 1" )
   END_RUNG
   RUNG wire#w4
      S_Coil( #Paso[2] )
   END_RUNG
   RUNG wire#w4
      R_Coil( #Marca[2] )
   END_RUNG
   RUNG wire#w4
      Coil( "Datos".Etiquetas.Reset )   // Resetea la Integracion del Caudal, para empezar a integrar nuevamente de 0.
   END_RUNG
   RUNG wire#w3
      S_Coil( #"Cinta 2" )
   END_RUNG
   RUNG wire#w3
      S_Coil( #"Cinta 3" )
   END_RUNG
   RUNG wire#w3
      R_Coil( #"Barrera 2" )
   END_RUNG
   RUNG wire#w2
      Contact( #SD031 )
      wire#w5
      R_Coil( #"Cinta 2" )   // En el caso del que la maquina de poner tapas no se haya desocupado no avanzara la caja.
   END_RUNG
   RUNG wire#w5
      S_Coil( #"Barrera 2" )
   END_RUNG
   // the same network as SCL:
   #_w1 := ((NOT #Parada AND #Marca[1]) OR (NOT #Parada AND #Paso[2])) AND #SD022 AND NOT #Flanco[9];   // rising edge of #SD022
   #Flanco[9] := #SD022;
   #_w2 := #_w1 AND NOT #SD031;
   #_w3 := #_w2 AND NOT #SD021;
   IF #_w3 THEN
       #"Barrera 1" := FALSE;
       #Marca[1] := FALSE;
       #"Cinta 1" := TRUE;
       #Paso[2] := TRUE;
       #Marca[2] := FALSE;
   END_IF;
   "Datos".Etiquetas.Reset := #_w3;   // Resetea la Integracion del Caudal, para empezar a integrar nuevamente de 0.
   IF #_w2 THEN
       #"Cinta 2" := TRUE;
       #"Cinta 3" := TRUE;
       #"Barrera 2" := FALSE;
   END_IF;
   IF #_w1 AND #SD031 THEN
       #"Cinta 2" := FALSE;   // En el caso del que la maquina de poner tapas no se haya desocupado no avanzara la caja.
       #"Barrera 2" := TRUE;
   END_IF;
END_REGION

REGION Network 6
   RUNG wire#powerrail
      I_Contact( #Parada )
      Contact( #Paso[2] )
      P_Contact(operand := #SD030, bit := #Flanco[7])
      I_Contact( #SD031 )
      wire#w1
      R_Coil( #"Cinta 3" )
   END_RUNG
   RUNG wire#w1
      S_Coil( #"Movimiento Eje Z 030" )
   END_RUNG
   // the same network as SCL:
   #_w1 := NOT #Parada AND #Paso[2] AND #SD030 AND NOT #Flanco[7];   // rising edge of #SD030
   #Flanco[7] := #SD030;
   IF #_w1 AND NOT #SD031 THEN
       #"Cinta 3" := FALSE;
       #"Movimiento Eje Z 030" := TRUE;
   END_IF;
END_REGION

REGION Network 7
   #_w1 := (NOT #Parada AND #Marca[3]) OR (NOT #Parada AND #Paso[2]);
   "Ton_ColocacionDeTapa".TON(IN := #_w1 AND #SD031, PT := T#500ms);
   IF "Ton_ColocacionDeTapa".Q THEN
       #"Succion 030" := FALSE;
       #"Movimiento Eje Z 030" := FALSE;
       #"Barrera 2" := FALSE;
       #"Cinta 3" := TRUE;
   END_IF;
   #_w2 := #_w1 AND #SD031 AND NOT #Flanco[6];   // rising edge of #SD031
   #Flanco[6] := #SD031;
   IF #_w2 THEN #"Succion 030" := TRUE; END_IF;
END_REGION

REGION Network 8
   RUNG wire#powerrail
      I_Contact( #Parada )
      Contact( #Marca[3] )
      wire#w1
      Contact( #SD032 )
      S_Coil( #Paso[3] )
   END_RUNG
   RUNG wire#powerrail
      I_Contact( #Parada )
      Contact( #Paso[2] )
   END_RUNG wire#w1
   // the same network as SCL:
   IF ((NOT #Parada AND #Marca[3]) OR (NOT #Parada AND #Paso[2])) AND #SD032 THEN #Paso[3] := TRUE; END_IF;
END_REGION

REGION Network 9
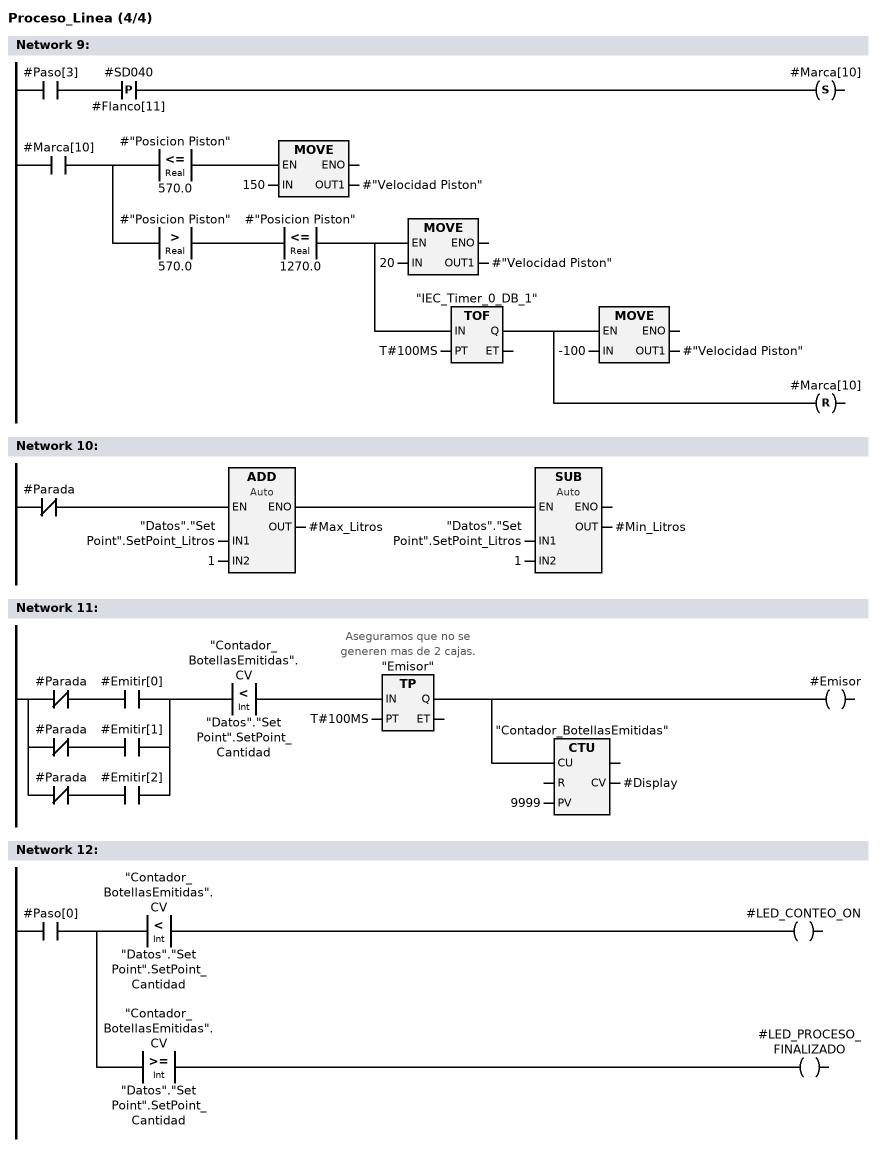
   #_w1 := #Paso[3] AND #SD040 AND NOT #Flanco[11];   // rising edge of #SD040
   #Flanco[11] := #SD040;
   IF #_w1 THEN #Marca[10] := TRUE; END_IF;
   IF #Marca[10] AND (#"Posicion Piston" <= 570.0) THEN #"Velocidad Piston" := 150; END_IF;
   #_w2 := #Marca[10] AND (#"Posicion Piston" > 570.0) AND (#"Posicion Piston" <= 1270.0);
   IF #_w2 THEN #"Velocidad Piston" := 20; END_IF;
   "IEC_Timer_0_DB_1".TOF(IN := #_w2, PT := T#100MS);
   IF "IEC_Timer_0_DB_1".Q THEN
       #"Velocidad Piston" := -100;
       #Marca[10] := FALSE;
   END_IF;
END_REGION

REGION Network 10
   RUNG wire#powerrail
      I_Contact( #Parada )
      Add(in1 := "Datos"."Set Point".SetPoint_Litros, in2 := 1, out => #Max_Litros)
      Sub(in1 := "Datos"."Set Point".SetPoint_Litros, in2 := 1, out => #Min_Litros)
   END_RUNG
   // the same network as SCL:
   IF NOT #Parada THEN
       #Max_Litros := "Datos"."Set Point".SetPoint_Litros + 1;
       #Min_Litros := "Datos"."Set Point".SetPoint_Litros - 1;
   END_IF;
END_REGION

REGION Network 11
   "Emisor".TP(IN := ((NOT #Parada AND #Emitir[0]) OR (NOT #Parada AND #Emitir[1]) OR (NOT #Parada AND #Emitir[2])) AND ("Contador_BotellasEmitidas".CV < "Datos"."Set Point".SetPoint_Cantidad),   // Aseguramos que no se generen mas de 2 cajas.
               PT := T#100MS);
   #Emisor := "Emisor".Q;
   "Contador_BotellasEmitidas".CTU(CU := "Emisor".Q, PV := 9999, CV => #Display);
END_REGION

REGION Network 12
   RUNG wire#powerrail
      Contact( #Paso[0] )
      wire#w1
      { S7_Templates := "SrcType := Int" } LT_Contact(in1 := "Contador_BotellasEmitidas".CV, in2 := "Datos"."Set Point".SetPoint_Cantidad)
      Coil( #LED_CONTEO_ON )
   END_RUNG
   RUNG wire#w1
      { S7_Templates := "SrcType := Int" } GE_Contact(in1 := "Contador_BotellasEmitidas".CV, in2 := "Datos"."Set Point".SetPoint_Cantidad)
      Coil( #LED_PROCESO_FINALIZADO )
   END_RUNG
   // the same network as SCL:
   #LED_CONTEO_ON := #Paso[0] AND ("Contador_BotellasEmitidas".CV < "Datos"."Set Point".SetPoint_Cantidad);
   #LED_PROCESO_FINALIZADO := #Paso[0] AND ("Contador_BotellasEmitidas".CV >= "Datos"."Set Point".SetPoint_Cantidad);
END_REGION
END_FUNCTION_BLOCK

FUNCTION "Arranque" : Void   // FC1, LAD
{ S7_Optimized_Access := 'TRUE' }
VERSION : 0.1
   VAR_TEMP   // added for the SCL form of the ladder/FBD networks
      _w1 : Bool;
   END_VAR
BEGIN

REGION Network 1
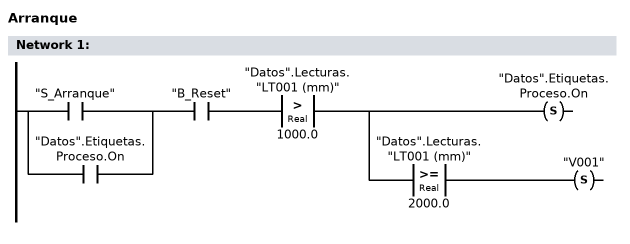
   RUNG wire#powerrail
      Contact( "S_Arranque" )
      wire#w1
      Contact( "B_Reset" )
      { S7_Templates := "SrcType := Real" } GT_Contact(in1 := "Datos".Lecturas."LT001 (mm)", in2 := 1000.0)
      wire#w2
      S_Coil( "Datos".Etiquetas.Proceso.On )
   END_RUNG
   RUNG wire#powerrail
      Contact( "Datos".Etiquetas.Proceso.On )
   END_RUNG wire#w1
   RUNG wire#w2
      { S7_Templates := "SrcType := Real" } GE_Contact(in1 := "Datos".Lecturas."LT001 (mm)", in2 := 2000.0)
      S_Coil( "V001" )
   END_RUNG
   // the same network as SCL:
   #_w1 := ("S_Arranque" OR "Datos".Etiquetas.Proceso.On) AND "B_Reset" AND ("Datos".Lecturas."LT001 (mm)" > 1000.0);
   IF #_w1 THEN "Datos".Etiquetas.Proceso.On := TRUE; END_IF;
   IF #_w1 AND ("Datos".Lecturas."LT001 (mm)" >= 2000.0) THEN "V001" := TRUE; END_IF;
END_REGION
END_FUNCTION

FUNCTION "Alarmas" : Void   // FC2, LAD
{ S7_Optimized_Access := 'TRUE' }
VERSION : 0.1
BEGIN

REGION Network 1
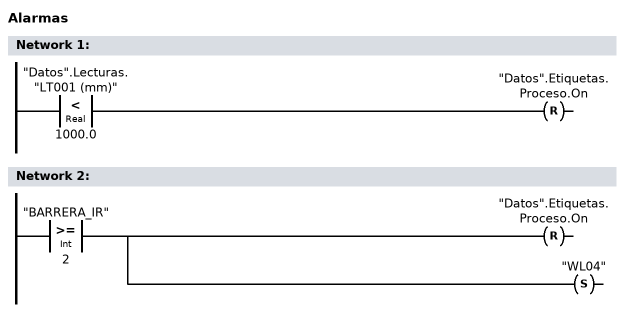
   RUNG wire#powerrail
      { S7_Templates := "SrcType := Real" } LT_Contact(in1 := "Datos".Lecturas."LT001 (mm)", in2 := 1000.0)
      R_Coil( "Datos".Etiquetas.Proceso.On )
   END_RUNG
   // the same network as SCL:
   IF "Datos".Lecturas."LT001 (mm)" < 1000.0 THEN "Datos".Etiquetas.Proceso.On := FALSE; END_IF;
END_REGION

REGION Network 2
   RUNG wire#powerrail
      { S7_Templates := "SrcType := Int" } GE_Contact(in1 := "BARRERA_IR", in2 := 2)
      wire#w1
      R_Coil( "Datos".Etiquetas.Proceso.On )
   END_RUNG
   RUNG wire#w1
      S_Coil( "WL04" )
   END_RUNG
   // the same network as SCL:
   IF "BARRERA_IR" >= 2 THEN
       "Datos".Etiquetas.Proceso.On := FALSE;
       "WL04" := TRUE;
   END_IF;
END_REGION
END_FUNCTION

FUNCTION "Escalado_AI" : Void   // FC3, LAD
{ S7_Optimized_Access := 'TRUE' }
VERSION : 0.1
   VAR_INPUT
      Sensor : Int;
      MAX_Sensor : Real;
      MIN_Sensor : Real;
      MAX_Canal : Int;
      MIN_Canal : Int;
   END_VAR
   VAR_OUTPUT
      Salida : Real;
   END_VAR
   VAR_TEMP
      Normalizado : Real;
   END_VAR
BEGIN

REGION Network 1
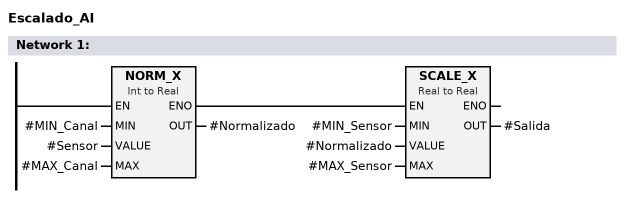
   RUNG wire#powerrail
      { S7_Templates := "[SrcType := Int, DestType := Real]" } Normalize(min := #MIN_Canal, value := #Sensor, max := #MAX_Canal, out => #Normalizado)
      { S7_Templates := "[SrcType := Real, DestType := Real]" } Scale(min := #MIN_Sensor, value := #Normalizado, max := #MAX_Sensor, out => #Salida)
   END_RUNG
   // the same network as SCL:
   #Normalizado := NORM_X(MIN := #MIN_Canal, VALUE := #Sensor, MAX := #MAX_Canal);
   #Salida := SCALE_X(MIN := #MIN_Sensor, VALUE := #Normalizado, MAX := #MAX_Sensor);
END_REGION
END_FUNCTION

FUNCTION "Escalado_AQ" : Void   // FC4, LAD
{ S7_Optimized_Access := 'TRUE' }
VERSION : 0.1
   VAR_INPUT
      Comando : Real;
      MAX_Comando : Real;
      MIN_Comando : Real;
      MAX_Actuador : Int;
      MIN_Actuador : Int;
   END_VAR
   VAR_OUTPUT
      Salida : Int;
   END_VAR
   VAR_TEMP
      Nomalizado : Real;
   END_VAR
BEGIN

REGION Network 1
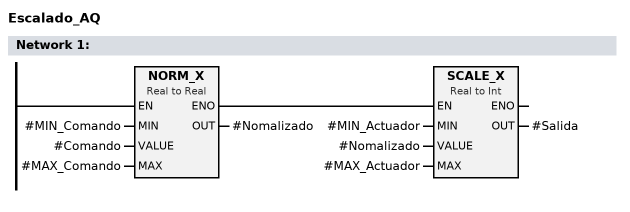
   RUNG wire#powerrail
      { S7_Templates := "[SrcType := Real, DestType := Real]" } Normalize(min := #MIN_Comando, value := #Comando, max := #MAX_Comando, out => #Nomalizado)
      { S7_Templates := "[SrcType := Real, DestType := Int]" } Scale(min := #MIN_Actuador, value := #Nomalizado, max := #MAX_Actuador, out => #Salida)
   END_RUNG
   // the same network as SCL:
   #Nomalizado := NORM_X(MIN := #MIN_Comando, VALUE := #Comando, MAX := #MAX_Comando);
   #Salida := SCALE_X(MIN := #MIN_Actuador, VALUE := #Nomalizado, MAX := #MAX_Actuador);
END_REGION
END_FUNCTION

FUNCTION "MHJ-PLC-Lab-Function-S71500" : Void   // FC9000, SCL
{ S7_Optimized_Access := 'TRUE' }
VERSION : 0.1
   VAR_TEMP
      Value : Byte;
      ForCounter : Int;
   END_VAR
   VAR CONSTANT
      Value_01_DW : DWord := 16#1223_5486;
      Value_02_DW : DWord := 16#A6C9_D1F5;
   END_VAR
BEGIN

   #Value:=PEEK(area := 16#82,
        dbNumber := 0,
        byteOffset := 511);
   #Value := #Value + 1;

   POKE(area := 16#82,
        dbNumber := 0,
        byteOffset := 511,
        value := #Value);

   POKE(area := 16#82,
        dbNumber := 0,
        byteOffset := 1016,
        value := #Value_01_DW);
   POKE(area := 16#82,
        dbNumber := 0,
        byteOffset := 1020,
        value := #Value_02_DW);

   FOR #ForCounter := 0 TO 63 DO
       #Value:=PEEK(area := 16#1,
            dbNumber := 0,
            byteOffset := #ForCounter);
       POKE(area := 16#81,
            dbNumber := 0,
            byteOffset := #ForCounter,
            value := #Value);
   END_FOR;
   #Value := PEEK(area := 16#1,
                  dbNumber := 0,
                  byteOffset := 512);
   POKE(area := 16#82,
        dbNumber := 0,
        byteOffset := 512,
        value := #Value);
END_FUNCTION

ORGANIZATION_BLOCK "Main"   // OB1, LAD, ProgramCycle
TITLE = "Main Program Sweep (Cycle)"
{ S7_Optimized_Access := 'TRUE' }
VERSION : 0.1
   VAR_INPUT
      Initial_Call : Bool;   // Initial call of this OB
      Remanence : Bool;   // =True, if remanent data are available
   END_VAR
BEGIN

REGION Network 1
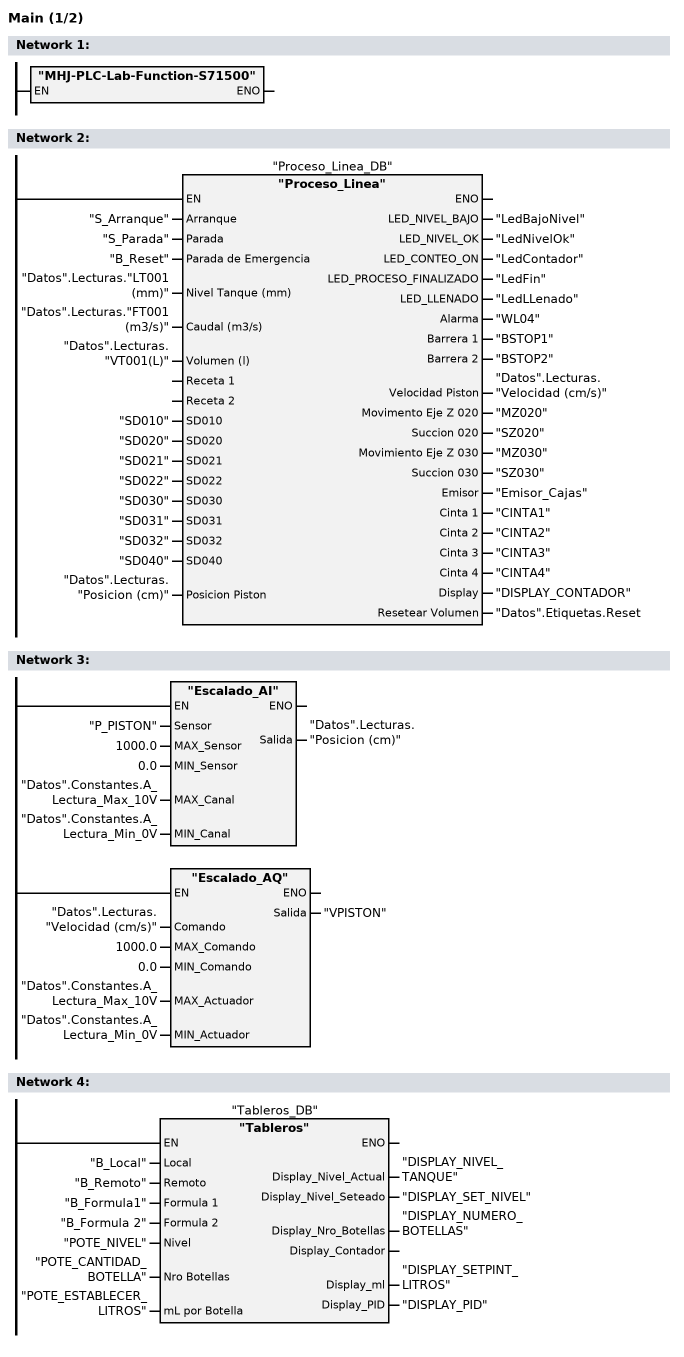
   RUNG wire#powerrail
      "MHJ-PLC-Lab-Function-S71500"()
   END_RUNG
   // the same network as SCL:
   "MHJ-PLC-Lab-Function-S71500"();
END_REGION

REGION Network 2
   RUNG wire#powerrail
      "Proceso_Linea_DB"(Arranque := "S_Arranque", Parada := "S_Parada", "Parada de Emergencia" := "B_Reset", "Nivel Tanque (mm)" := "Datos".Lecturas."LT001 (mm)", "Caudal (m3/s)" := "Datos".Lecturas."FT001 (m3/s)", "Volumen (l)" := "Datos".Lecturas."VT001(L)", "Receta 1" :=, "Receta 2" :=, SD010 := "SD010", SD020 := "SD020", SD021 := "SD021", SD022 := "SD022", SD030 := "SD030", SD031 := "SD031", SD032 := "SD032", SD040 := "SD040", "Posicion Piston" := "Datos".Lecturas."Posicion (cm)", LED_NIVEL_BAJO => "LedBajoNivel", LED_NIVEL_OK => "LedNivelOk", LED_CONTEO_ON => "LedContador", LED_PROCESO_FINALIZADO => "LedFin", LED_LLENADO => "LedLLenado", Alarma => "WL04", "Barrera 1" => "BSTOP1", "Barrera 2" => "BSTOP2", "Velocidad Piston" => "Datos".Lecturas."Velocidad (cm/s)", "Movimento Eje Z 020" => "MZ020", "Succion 020" => "SZ020", "Movimiento Eje Z 030" => "MZ030", "Succion 030" => "SZ030", Emisor => "Emisor_Cajas", "Cinta 1" => "CINTA1", "Cinta 2" => "CINTA2", "Cinta 3" => "CINTA3", "Cinta 4" => "CINTA4", Display => "DISPLAY_CONTADOR", "Resetear Volumen" => "Datos".Etiquetas.Reset)
   END_RUNG
   // the same network as SCL:
   "Proceso_Linea_DB"(Arranque := "S_Arranque",   // "Proceso_Linea"
                      Parada := "S_Parada",
                      "Parada de Emergencia" := "B_Reset",
                      "Nivel Tanque (mm)" := "Datos".Lecturas."LT001 (mm)",
                      "Caudal (m3/s)" := "Datos".Lecturas."FT001 (m3/s)",
                      "Volumen (l)" := "Datos".Lecturas."VT001(L)",
                      SD010 := "SD010",
                      SD020 := "SD020",
                      SD021 := "SD021",
                      SD022 := "SD022",
                      SD030 := "SD030",
                      SD031 := "SD031",
                      SD032 := "SD032",
                      SD040 := "SD040",
                      "Posicion Piston" := "Datos".Lecturas."Posicion (cm)",
                      LED_NIVEL_BAJO => "LedBajoNivel",
                      LED_NIVEL_OK => "LedNivelOk",
                      LED_CONTEO_ON => "LedContador",
                      LED_PROCESO_FINALIZADO => "LedFin",
                      LED_LLENADO => "LedLLenado",
                      Alarma => "WL04",
                      "Barrera 1" => "BSTOP1",
                      "Barrera 2" => "BSTOP2",
                      "Velocidad Piston" => "Datos".Lecturas."Velocidad (cm/s)",
                      "Movimento Eje Z 020" => "MZ020",
                      "Succion 020" => "SZ020",
                      "Movimiento Eje Z 030" => "MZ030",
                      "Succion 030" => "SZ030",
                      Emisor => "Emisor_Cajas",
                      "Cinta 1" => "CINTA1",
                      "Cinta 2" => "CINTA2",
                      "Cinta 3" => "CINTA3",
                      "Cinta 4" => "CINTA4",
                      Display => "DISPLAY_CONTADOR",
                      "Resetear Volumen" => "Datos".Etiquetas.Reset);
END_REGION

REGION Network 3
   RUNG wire#powerrail
      "Escalado_AI"(Sensor := "P_PISTON", MAX_Sensor := 1000.0, MIN_Sensor := 0.0, MAX_Canal := "Datos".Constantes.A_Lectura_Max_10V, MIN_Canal := "Datos".Constantes.A_Lectura_Min_0V, Salida => "Datos".Lecturas."Posicion (cm)")
   END_RUNG
   RUNG wire#powerrail
      "Escalado_AQ"(Comando := "Datos".Lecturas."Velocidad (cm/s)", MAX_Comando := 1000.0, MIN_Comando := 0.0, MAX_Actuador := "Datos".Constantes.A_Lectura_Max_10V, MIN_Actuador := "Datos".Constantes.A_Lectura_Min_0V, Salida => "VPISTON")
   END_RUNG
   // the same network as SCL:
   "Escalado_AI"(Sensor := "P_PISTON",
                 MAX_Sensor := 1000.0,
                 MIN_Sensor := 0.0,
                 MAX_Canal := "Datos".Constantes.A_Lectura_Max_10V,
                 MIN_Canal := "Datos".Constantes.A_Lectura_Min_0V,
                 Salida => "Datos".Lecturas."Posicion (cm)");
   "Escalado_AQ"(Comando := "Datos".Lecturas."Velocidad (cm/s)",
                 MAX_Comando := 1000.0,
                 MIN_Comando := 0.0,
                 MAX_Actuador := "Datos".Constantes.A_Lectura_Max_10V,
                 MIN_Actuador := "Datos".Constantes.A_Lectura_Min_0V,
                 Salida => "VPISTON");
END_REGION

REGION Network 4
   RUNG wire#powerrail
      "Tableros_DB"(Local := "B_Local", Remoto := "B_Remoto", "Formula 1" := "B_Formula1", "Formula 2" := "B_Formula 2", Nivel := "POTE_NIVEL", "Nro Botellas" := "POTE_CANTIDAD_BOTELLA", "mL por Botella" := "POTE_ESTABLECER_LITROS", Display_Nivel_Actual => "DISPLAY_NIVEL_TANQUE", Display_Nivel_Seteado => "DISPLAY_SET_NIVEL", Display_Nro_Botellas => "DISPLAY_NUMERO_BOTELLAS", Display_Contador =>, Display_ml => "DISPLAY_SETPINT_LITROS", Display_PID => "DISPLAY_PID")
   END_RUNG
   // the same network as SCL:
   "Tableros_DB"(Local := "B_Local",   // "Tableros"
                 Remoto := "B_Remoto",
                 "Formula 1" := "B_Formula1",
                 "Formula 2" := "B_Formula 2",
                 Nivel := "POTE_NIVEL",
                 "Nro Botellas" := "POTE_CANTIDAD_BOTELLA",
                 "mL por Botella" := "POTE_ESTABLECER_LITROS",
                 Display_Nivel_Actual => "DISPLAY_NIVEL_TANQUE",
                 Display_Nivel_Seteado => "DISPLAY_SET_NIVEL",
                 Display_Nro_Botellas => "DISPLAY_NUMERO_BOTELLAS",
                 Display_ml => "DISPLAY_SETPINT_LITROS",
                 Display_PID => "DISPLAY_PID");
END_REGION

REGION Network 5
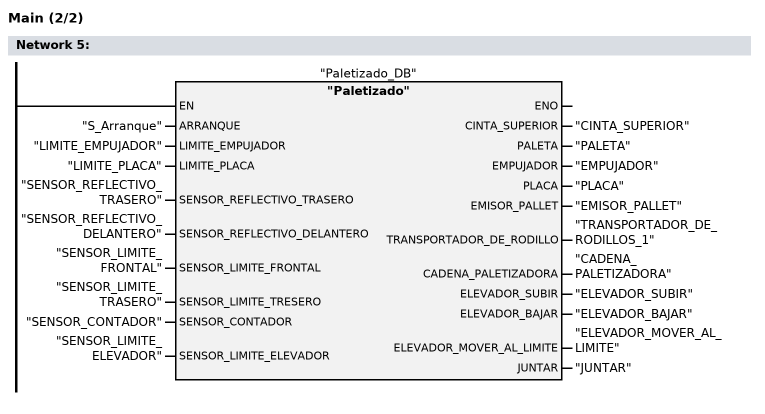
   RUNG wire#powerrail
      "Paletizado_DB"(ARRANQUE := "S_Arranque", LIMITE_EMPUJADOR := "LIMITE_EMPUJADOR", LIMITE_PLACA := "LIMITE_PLACA", SENSOR_REFLECTIVO_TRASERO := "SENSOR_REFLECTIVO_TRASERO", SENSOR_REFLECTIVO_DELANTERO := "SENSOR_REFLECTIVO_DELANTERO", SENSOR_LIMITE_FRONTAL := "SENSOR_LIMITE_FRONTAL", SENSOR_LIMITE_TRESERO := "SENSOR_LIMITE_TRASERO", SENSOR_CONTADOR := "SENSOR_CONTADOR", SENSOR_LIMITE_ELEVADOR := "SENSOR_LIMITE_ELEVADOR", CINTA_SUPERIOR => "CINTA_SUPERIOR", PALETA => "PALETA", EMPUJADOR => "EMPUJADOR", PLACA => "PLACA", EMISOR_PALLET => "EMISOR_PALLET", TRANSPORTADOR_DE_RODILLO => "TRANSPORTADOR_DE_RODILLOS_1", CADENA_PALETIZADORA => "CADENA_PALETIZADORA", ELEVADOR_SUBIR => "ELEVADOR_SUBIR", ELEVADOR_BAJAR => "ELEVADOR_BAJAR", ELEVADOR_MOVER_AL_LIMITE => "ELEVADOR_MOVER_AL_LIMITE", JUNTAR => "JUNTAR")
   END_RUNG
   // the same network as SCL:
   "Paletizado_DB"(ARRANQUE := "S_Arranque",   // "Paletizado"
                   LIMITE_EMPUJADOR := "LIMITE_EMPUJADOR",
                   LIMITE_PLACA := "LIMITE_PLACA",
                   SENSOR_REFLECTIVO_TRASERO := "SENSOR_REFLECTIVO_TRASERO",
                   SENSOR_REFLECTIVO_DELANTERO := "SENSOR_REFLECTIVO_DELANTERO",
                   SENSOR_LIMITE_FRONTAL := "SENSOR_LIMITE_FRONTAL",
                   SENSOR_LIMITE_TRESERO := "SENSOR_LIMITE_TRASERO",
                   SENSOR_CONTADOR := "SENSOR_CONTADOR",
                   SENSOR_LIMITE_ELEVADOR := "SENSOR_LIMITE_ELEVADOR",
                   CINTA_SUPERIOR => "CINTA_SUPERIOR",
                   PALETA => "PALETA",
                   EMPUJADOR => "EMPUJADOR",
                   PLACA => "PLACA",
                   EMISOR_PALLET => "EMISOR_PALLET",
                   TRANSPORTADOR_DE_RODILLO => "TRANSPORTADOR_DE_RODILLOS_1",
                   CADENA_PALETIZADORA => "CADENA_PALETIZADORA",
                   ELEVADOR_SUBIR => "ELEVADOR_SUBIR",
                   ELEVADOR_BAJAR => "ELEVADOR_BAJAR",
                   ELEVADOR_MOVER_AL_LIMITE => "ELEVADOR_MOVER_AL_LIMITE",
                   JUNTAR => "JUNTAR");
END_REGION
END_ORGANIZATION_BLOCK

ORGANIZATION_BLOCK "Cyclic_Int_PID"   // OB30, LAD, CyclicInterrupt
{ S7_Optimized_Access := 'TRUE' }
VERSION : 0.1
   VAR_INPUT
      Initial_Call : Bool;   // Initial call of this OB
      Event_Count : Int;   // Events discarded
   END_VAR
BEGIN

REGION Network 1
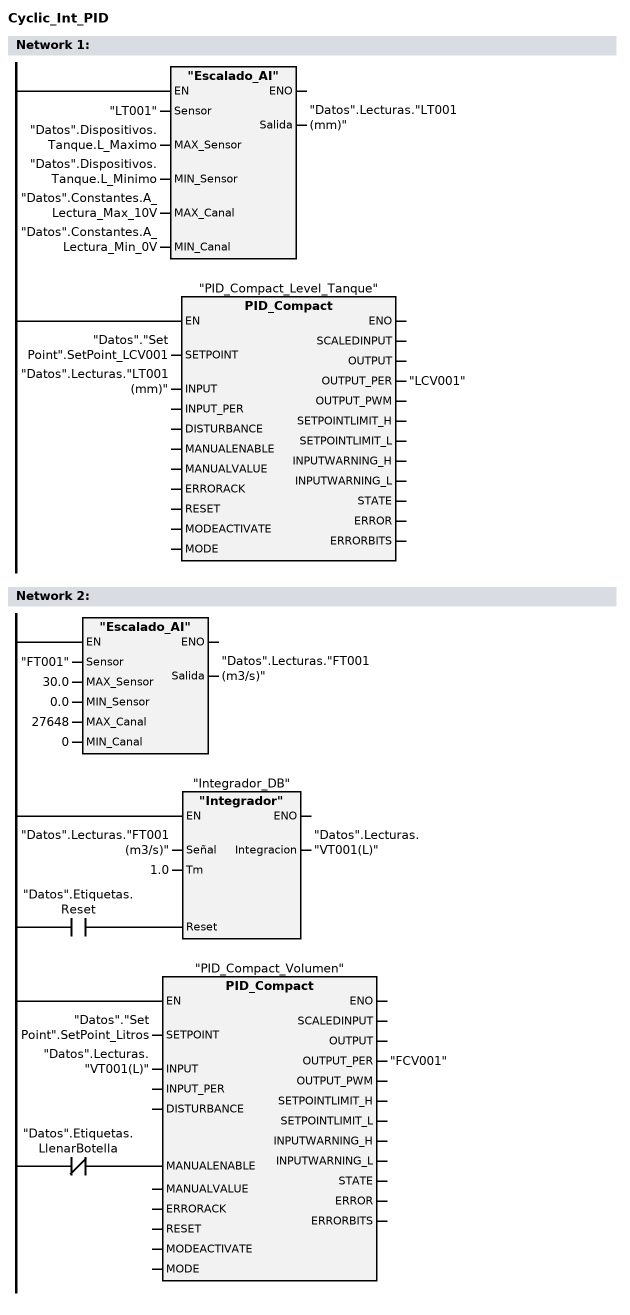
   "Escalado_AI"(Sensor := "LT001",
                 MAX_Sensor := "Datos".Dispositivos.Tanque.L_Maximo,
                 MIN_Sensor := "Datos".Dispositivos.Tanque.L_Minimo,
                 MAX_Canal := "Datos".Constantes.A_Lectura_Max_10V,
                 MIN_Canal := "Datos".Constantes.A_Lectura_Min_0V,
                 Salida => "Datos".Lecturas."LT001 (mm)");
   "PID_Compact_Level_Tanque"(Setpoint := "Datos"."Set Point".SetPoint_LCV001,   // PID_Compact
                           Input := "Datos".Lecturas."LT001 (mm)",
                           Output_PER => "LCV001");
END_REGION

REGION Network 2
   "Escalado_AI"(Sensor := "FT001",
                 MAX_Sensor := 30.0,
                 MIN_Sensor := 0.0,
                 MAX_Canal := 27648,
                 MIN_Canal := 0,
                 Salida => "Datos".Lecturas."FT001 (m3/s)");
   "Integrador_DB"(Señal := "Datos".Lecturas."FT001 (m3/s)",   // "Integrador"
                   Tm := 1.0,
                   Reset := "Datos".Etiquetas.Reset,
                   Integracion => "Datos".Lecturas."VT001(L)");
   "PID_Compact_Volumen"(Setpoint := "Datos"."Set Point".SetPoint_Litros,   // PID_Compact
                         Input := "Datos".Lecturas."VT001(L)",
                         ManualEnable := NOT "Datos".Etiquetas.LlenarBotella,
                         Output_PER => "FCV001");
END_REGION
END_ORGANIZATION_BLOCK